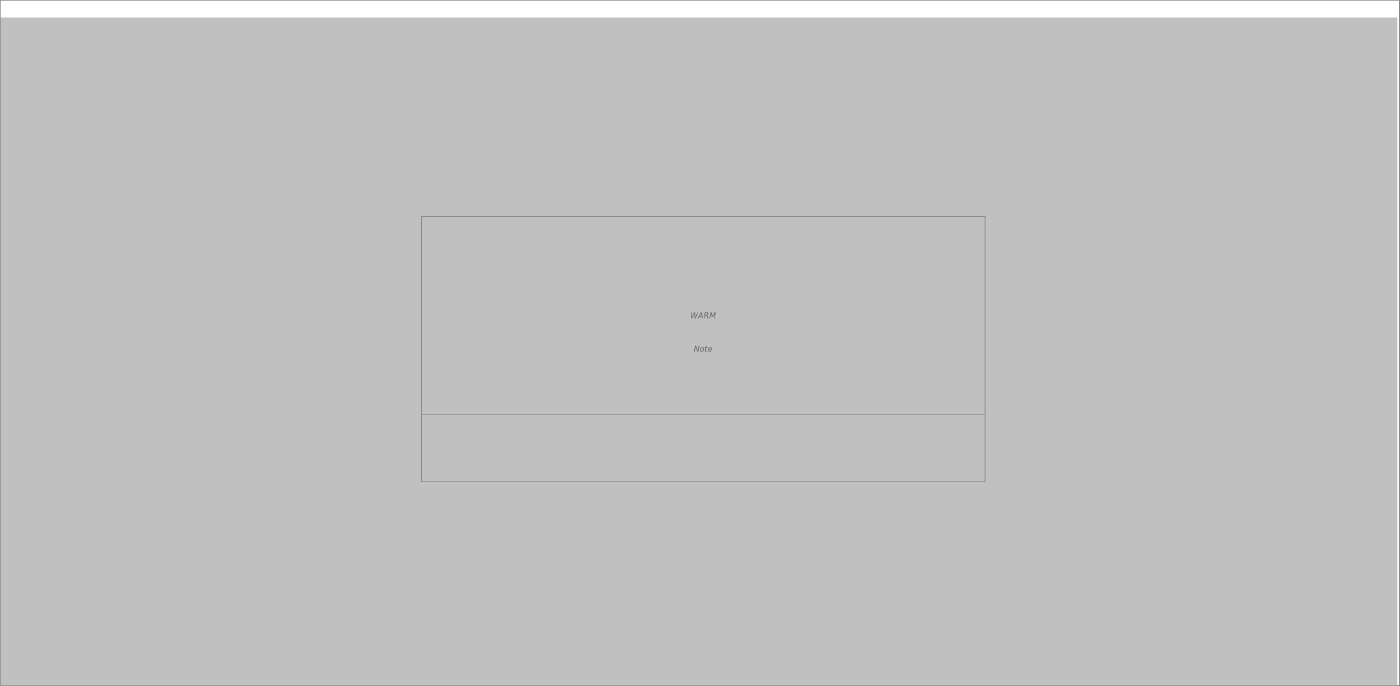
VISUALIZATION Manual  // 1755x860
    TabControl (0,0 1755x860), input disabled if: gWarmShowHMI.showFlag or gNoteShowHMI.showFlag or gPDVOpencondition or S_PDVSafeCtr.busy or gSPOUBusy
        shows Overview()
        shows Overview_Total()
        [0]: TabTitle=All Show
        [1]: TabTitle=Part Show
    Rectangle (0,22 1751x838), invisible if: (Not gWarmShowHMI.showFlag and Not gNoteShowHMI.showFlag) or gCtrlMode=ControlMode.eAutoCtrMode
    Frame (528,271 707x249), invisible if: NOT gWarmShowHMI.showFlag
        shows WARM(warmHMI := gWarmShowHMI)
    Frame (528,271 707x333), invisible if: Not gNoteShowHMI.showFlag or gCtrlMode=ControlMode.eAutoCtrMode
        shows Note(noteHMI := gNoteShowHMI)
END_VISUALIZATION

(* stored: Version 1.1.0.1, ProductVersion 3.1.4024.12
   Visu Manual: Id {75863b09-3105-497d-b5d0-aa0de1e2a49c} *)
